// TIA Portal V17 export
// export: Created 2024-08-29T18:23:44.3707262Z, ExportSetting WithDefaults, DisplayName Totally Integrated Automation Portal, DisplayVersion V17 Update 7, DisplayName TIA Portal Openness, DisplayVersion V17 Update 7, DisplayName TIA Portal Version Control Interface, DisplayVersion V17, DisplayName SINAMICS Startdrive Advanced, DisplayVersion V17 SP2, DisplayName SINAMICS Startdrive G110M, G120, G120C, G120D, G120P, G115D, DisplayVersion V17 SP2, DisplayName SINAMICS Startdrive G130, G150, S120, S150, SINAMICS MV, S210, DisplayVersion V17 SP2, DisplayName STEP 7 Professional, DisplayVersion V17 Update 7, DisplayName STEP 7 Safety, DisplayVersion V17 Update 6, DisplayName WinCC Advanced / Unified PC, DisplayVersion V17 Update 7
DATA_BLOCK "step"   // DB4
{ S7_Optimized_Access := 'TRUE' }
VERSION : 0.1
// stored: AutoNumber false, DBAccessibleFromOPCUA true, DBAccessibleFromWebserver true, IsOnlyStoredInLoadMemory false, IsRetainMemResEnabled false, IsWriteProtectedInAS false, MemoryReserve 100
   VAR RETAIN
      "time" : Array[0..32, 0..25] of Int;   // Tiempo de duración de cada paso [modelo, paso]
      number : Array[0..32] of Int;   // Número de pasos por modelo
   END_VAR
   VAR
      stepChangeTimer : DInt := 0;
      stepChangeTimerStart : Bool := FALSE;
      counterDone : Bool := FALSE;
   END_VAR
BEGIN
   "time"[0,0] := 0;
   "time"[0,1..5] := 500;
   "time"[0,6] := 1000;
   "time"[0,7] := 500;
   "time"[0,8] := 1000;
   "time"[0,9..10] := 500;
   "time"[0,11..25] := 0;
   "time"[1,0] := 0;
   "time"[1,1..5] := 500;
   "time"[1,6] := 1000;
   "time"[1,7] := 500;
   "time"[1,8] := 1000;
   "time"[1,9..10] := 500;
   "time"[1,11..25] := 0;
   "time"[2,0] := 0;
   "time"[2,1..5] := 500;
   "time"[2,6] := 1000;
   "time"[2,7] := 500;
   "time"[2,8] := 1000;
   "time"[2,9..10] := 500;
   "time"[2,11..25] := 0;
   "time"[3,0] := 0;
   "time"[3,1] := 500;
   "time"[3,2..4] := 1500;
   "time"[3,5..11] := 500;
   "time"[3,12..25] := 0;
   "time"[4,0] := 0;
   "time"[4,1] := 500;
   "time"[4,2..4] := 1500;
   "time"[4,5..11] := 500;
   "time"[4,12..25] := 0;
   "time"[5,0] := 0;
   "time"[5,1] := 1000;
   "time"[5,2] := 0;
   "time"[5,3] := 1000;
   "time"[5,4..25] := 0;
   "time"[6,0] := 0;
   "time"[6,1..2] := 1500;
   "time"[6,3] := 0;
   "time"[6,4..9] := 3000;
   "time"[6,10..25] := 0;
   "time"[7,0] := 0;
   "time"[7,1..2] := 1500;
   "time"[7,3] := 0;
   "time"[7,4..9] := 3000;
   "time"[7,10..25] := 0;
   "time"[8,0] := 0;
   "time"[8,1..2] := 1500;
   "time"[8,3] := 0;
   "time"[8,4..9] := 3000;
   "time"[8,10..25] := 0;
   "time"[9,0..3] := 0;
   "time"[9,4..5] := 500;
   "time"[9,6..25] := 0;
   "time"[10,0..3] := 0;
   "time"[10,4..5] := 500;
   "time"[10,6..25] := 0;
   "time"[11,0..3] := 0;
   "time"[11,4..5] := 500;
   "time"[11,6..25] := 0;
   "time"[12,0..3] := 0;
   "time"[12,4..5] := 500;
   "time"[12,6..25] := 0;
   "time"[13,0..3] := 0;
   "time"[13,4..5] := 500;
   "time"[13,6..25] := 0;
   "time"[14,0..3] := 0;
   "time"[14,4..5] := 500;
   "time"[14,6..25] := 0;
   "time"[15,0..25] := 0;
   "time"[16,0..3] := 0;
   "time"[16,4..5] := 500;
   "time"[16,6..25] := 0;
   "time"[17,0..3] := 0;
   "time"[17,4..5] := 500;
   "time"[17,6..25] := 0;
   "time"[18,0..3] := 0;
   "time"[18,4..5] := 500;
   "time"[18,6..25] := 0;
   "time"[19,0..3] := 0;
   "time"[19,4..5] := 500;
   "time"[19,6..25] := 0;
   "time"[20,0..25] := 0;
   "time"[21,0..25] := 0;
   "time"[22,0..25] := 0;
   "time"[23,0..25] := 0;
   "time"[24,0..25] := 0;
   "time"[25,0..25] := 0;
   "time"[26,0..25] := 0;
   "time"[27,0..25] := 0;
   "time"[28,0..25] := 0;
   "time"[29,0..25] := 0;
   "time"[30,0..25] := 0;
   "time"[31,0..25] := 0;
   "time"[32,0..25] := 0;
   number[0..2] := 10;
   number[3..4] := 11;
   number[5] := 3;
   number[6..14] := 9;
   number[15] := 8;
   number[16..19] := 9;
   number[20..32] := 0;
END_DATA_BLOCK
